FUNCTION_BLOCK E_REND_2 (* Rendezvous (AND) of two events *)
  (* Standard: 61499-2 *)
  (* Version 1.0, 2025-01-07, david *)
  PACKAGE dinasore::events;
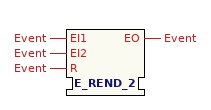
  EVENT_INPUT
    EI1; (* first event to wait for *)
    EI2; (* second event to wait for *)
    R; (* reset the FB to inital state (i.e., wait again for both events) *)
  END_EVENT
  EVENT_OUTPUT
    EO; (* triggered when both EI1 and EI2 occured at least once *)
  END_EVENT
END_FUNCTION_BLOCK
